(* CoDeSys 2.3 export: LOGICSENSCLASS.EXP *)

(* Data type in ENUM *)
TYPE LogicSensClass : (LogicalIn:=1, LogicalInverter, LogicalComposer, LogicalAdapter);
END_TYPE
